// TIA Portal V16 export
// export: Created 2021-12-08T09:54:17.4565558Z, ExportSetting None, DisplayName Totally Integrated Automation Portal, DisplayVersion V16, DisplayName TIA Portal Version Control Interface, DisplayVersion V16, DisplayName TIA Portal Openness, DisplayVersion V16, DisplayName STEP 7 Professional, DisplayVersion V16, DisplayName STEP 7 Safety, DisplayVersion V16, DisplayName WinCC Advanced, DisplayVersion V16
FUNCTION "CommentTest" : Void   // FC4, LAD
{ S7_Optimized_Access := 'TRUE' }
// stored: SetENOAutomatically false
   VAR_INPUT
      Input1 : Bool;   // WOW! UN COMMENTO :D / WOW! A COMMENT c:
   END_VAR
   VAR_OUTPUT
      Output1 : Bool;
   END_VAR
   VAR_IN_OUT
      TrigInOut_1 : Bool;
      TrigInOut_2 : Bool;
      InOut : Bool;
   END_VAR
   VAR_TEMP   // added for the SCL form of the ladder/FBD networks
      _w1 : Bool;
      _w2 : Bool;
   END_VAR
BEGIN

REGION Network 1
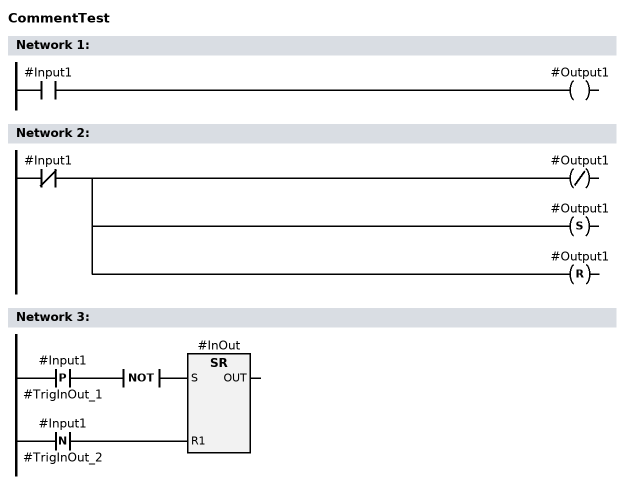
   RUNG wire#powerrail
      Contact( #Input1 )
      Coil( #Output1 )
   END_RUNG
   // the same network as SCL:
   #Output1 := #Input1;
END_REGION

REGION Network 2
   RUNG wire#powerrail
      I_Contact( #Input1 )
      wire#w1
      I_Coil( #Output1 )
   END_RUNG
   RUNG wire#w1
      S_Coil( #Output1 )
   END_RUNG
   RUNG wire#w1
      R_Coil( #Output1 )
   END_RUNG
   // the same network as SCL:
   #Output1 := NOT (NOT #Input1);
   IF NOT #Input1 THEN
       #Output1 := TRUE;
       #Output1 := FALSE;
   END_IF;
END_REGION

REGION Network 3
   RUNG wire#powerrail
      P_Contact(operand := #Input1, bit := #TrigInOut_1)
      Not()
      S_SR(operand := #InOut, r1 := wire#w1)
   END_RUNG
   RUNG wire#powerrail
      N_Contact(operand := #Input1, bit := #TrigInOut_2)
   END_RUNG wire#w1
   // the same network as SCL:
   #_w1 := #Input1 AND NOT #TrigInOut_1;   // rising edge of #Input1
   #TrigInOut_1 := #Input1;
   #_w2 := NOT #Input1 AND #TrigInOut_2;   // falling edge of #Input1
   #TrigInOut_2 := #Input1;
   IF NOT #_w1 THEN
       #InOut := TRUE;   // SR flip-flop
   END_IF;
   IF #_w2 THEN #InOut := FALSE; END_IF;
END_REGION
END_FUNCTION
